// TIA Portal V20 export
DATA_BLOCK "process_DB"   // DB1
// stored: MemoryReserve 100, Namespace ELY_1
BEGIN
END_DATA_BLOCK
